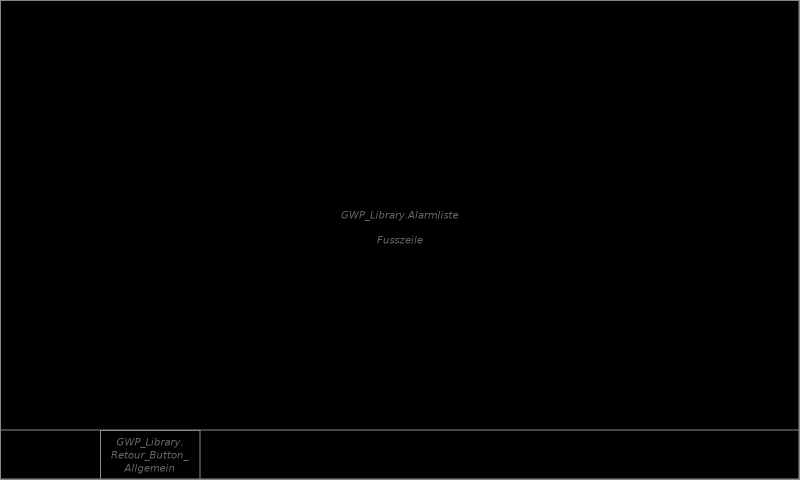
VISUALIZATION Alarmliste  // 800x480
    Frame (0,0 800x430)
        shows GWP_Library.Alarmliste()
    Frame (0,0 800x480)
        shows Fusszeile()
    Frame (100,430 100x50)
        shows GWP_Library.Retour_Button_Allgemein()
END_VISUALIZATION

(* stored: Version 1.1.0.1, ProductVersion 3.1.4022.6
   Visu Alarmliste: Id {54bcf857-3264-4d79-a74e-6ec6abdf9a48} *)
